(* IEC 61131-3 sources: Lasal/CPU_5344_V01/Class/Logic_And_4, 1 file *)

(* ---- Logic_And_4.st ---- *)
(*!
<Class
	Name               = "Logic_And_4"
	Revision           = "1.2"
	RealtimeTask       = "false"
	CyclicTask         = "false"
	BackgroundTask     = "false"
	Sigmatek           = "true"
	OSInterface        = "false"
	HighPriority       = "false"
	Automatic          = "false"
	UpdateMode         = "Prescan"
	IconPath           = ".\Class\Logic_And_4\Logic_And_Base.ico"
	SharedCommandTable = "true"
	Objectsize         = "(284,120)"
	Comment            = "V1.2 Logic AND class with 4 operands">
	<Channels>
		<Server
			Name           = "result"
			Initialize     = "false"
			Visualized     = "true"
			WriteProtected = "true"
			Comment        = "result of the calculation of operand1 - operand4">
		</Server>
		<Client Name="Op1" Required="false" Internal="false" Comment="Operand 1"/>
		<Client Name="Op2" Required="false" Internal="false" Comment="Operand 2"/>
		<Client Name="Op3" Required="false" Internal="false" Comment="Operand 3"/>
		<Client Name="Op4" Required="false" Internal="false" Comment="Operand 4"/>
	</Channels>
	<Network Name="Logic_And_4">
		<!-- List of Components in this network -->
		<Components>
			<Object
				Name       = "_base"
				Class      = "Logic_And_Base"
				Position   = "(660,540)"
				Visualized = "true">
				<Channels>
					<Server Name="result"/>
				</Channels>
			</Object>
		</Components>
		<Comments>
		</Comments>
		<!-- List of Connections in this network -->
		<Connections>
			<Connection Source="this.result" Destination="_base.result" Vertices="(1132,210),(960,630),"/>
		</Connections>
		<!-- Headerfiles -->
		<Options>
		</Options>
	</Network>
</Class>
*)
#pragma using Logic_And_Base

Logic_And_4 : CLASS
: Logic_And_Base
  //Servers:
  //Clients:
	Op1 	: CltCh_DINT;
	Op2 	: CltCh_DINT;
	Op3 	: CltCh_DINT;
	Op4 	: CltCh_DINT;
  //Variables:
  //Functions:
  //Tables:
	FUNCTION @STD
		VAR_OUTPUT
			ret_code	: CONFSTATES;
		END_VAR;
	FUNCTION GLOBAL TAB @CT_;
END_CLASS;
